FUNCTION_BLOCK FB_CartCtrlStandColuAdjust EXTENDS FB_CartCtrlBase
VAR_INPUT
END_VAR
VAR_OUTPUT
END_VAR
VAR

	m_actJntPos: Vec8d;
	m_tarJntPos : LREAL;
	m_trjJntPos : LREAL;
	m_trjJntInc : LREAL;
	m_lastTrajJntPos : LREAL;
	m_initActJntPos: LREAL;
	m_maxJntPos : vec8d;

	// time threshold to 5-8joint after it's enabled
	m_cartAdjustStartWaitTime :LREAL := 0.3;
	
	//adjust start  time 
	m_adjustStartTime :LREAL;
	m_jntOTG : FB_secOrdTrajFilter;
	
	// filter cut-off frequency for joint 3 velocity
	m_cmdJoystickLpfJnt3Freq : LREAL :=8;
	m_cartCtrlFreq :LREAL:=8000;
END_VAR

// override this function in each exact controller
METHOD PROTECTED calcCmdJntPos : BOOL
VAR_IN_OUT CONSTANT
	// slave cart joint data
	i_slaveCart :FB_SlaveCart;
END_VAR

VAR
	i:INT;
END_VAR
//In this method, 5 represents the pillar postion , 6 represents the beam rotation angle ,7 represents the beam stretch position ,8 represents the overhang angle
m_adjustStartTime :=LIMIT(0, m_adjustStartTime + g_cartCtrlCycleTime, 1);
m_actJntPos := i_slaveCart.curJntPos;
m_jntEnableFlag[5] := BOOL_TO_INT( NOT SafetyCheck.m_safetyCheckData.m_cartStandColumnErr);

IF m_adjustStartTime > m_cartAdjustStartWaitTime THEN
	m_trjJntInc := m_trjJntInc + (i_slaveCart.m_columnJntVel * g_cartCtrlCycleTime);
	m_trjJntPos := m_initActJntPos + m_trjJntInc;
	m_jntPosReachLimit[5] := calcCmdReachLimit();
	m_tarJntPos := LIMIT(GVL_CartMotorParameters.g_minJntPos[5] + GVL_CartControlParameters.g_carJntSoftwareLimit[5], m_trjJntPos, MAX(m_actJntPos[5],i_slaveCart.m_cartDataFromUI.m_standColumnHightLimit));
	m_jntOTG.run(i_targetPos:= m_tarJntPos, i_targetVel:= 0.0, o_cmdAcc=> , o_cmdVel=> , o_cmdPos=>m_cmdJntPos[5] );
END_IF
END_METHOD

METHOD calcCmdReachLimit : BOOL
VAR_INPUT
END_VAR

VAR
	i : INT;
END_VAR

IF (GVL_CartMotorParameters.g_minJntPos[5] + GVL_CartControlParameters.g_carJntSoftwareLimit[5]) >= m_trjJntPos THEN
	IF (m_trjJntInc - m_lastTrajJntPos) <0 THEN
		m_trjJntInc := m_lastTrajJntPos;
	END_IF
	calcCmdReachLimit := TRUE;

ELSIF m_trjJntPos>=(m_maxJntPos[5] - GVL_CartControlParameters.g_carJntSoftwareLimit[5]) THEN
	IF (m_trjJntInc - m_lastTrajJntPos) >0 THEN
		m_trjJntInc := m_lastTrajJntPos;
	END_IF
	calcCmdReachLimit := TRUE;
END_IF
m_lastTrajJntPos := m_trjJntInc;
END_METHOD

// override this function in each exact controller
// NOTICE: set joint control mode here, and do some initialization if needed
METHOD PUBLIC init : BOOL
VAR_IN_OUT CONSTANT
	i_slaveCart	:FB_SlaveCart;
END_VAR
VAR_IN_OUT 
	r_cartCtrlCmd :ST_SlaveArmCtrlCmds;
END_VAR
VAR
	i:INT;
END_VAR
// check if to hold the command joint position unchanged
//m_holdLastCmds := checkToHoldLastCmds(i_slaveCart);
m_holdLastCmds := checkToHoldLastCmds(i_slaveCart);
SUPER^.init(i_slaveCart,r_cartCtrlCmd);
m_cmdJntPos[5]:=i_slaveCart.m_curJntPos[5];

m_jntEnableFlag[5] := BOOL_TO_INT( NOT SafetyCheck.m_safetyCheckData.m_cartStandColumnErr);
m_jntOPMode[5]:= DriverOPMode_cspMZ;
IF GVL_interactUI.g_heightLimitEnbale=FALSE THEN
	m_maxJntPos[5] := i_slaveCart.m_cartDataFromUI.m_standColumnHightLimit;
ELSE
	m_maxJntPos[5] := i_slaveCart.m_cartDataFromUI.m_standColumnHightLimit + GVL_CartControlParameters.g_carJntSoftwareLimit[5];
END_IF
m_initActJntPos:=m_cmdJntPos[5];
m_jntOTG.init(i_curCmdPos:= m_cmdJntPos[5], i_curCmdVel:= 0, i_maxV:=GVL_CartControlParameters.g_maxJntVel[5] , i_maxA:=GVL_CartControlParameters.g_maxJntAcc[5] , i_Ts:=g_cartCtrlCycleTime );

m_trjJntInc := 0;
m_lastTrajJntPos := 0;
m_adjustStartTime := 0;
// update commands to arm
copyCmds(r_cartCtrlCmd);
END_METHOD

END_FUNCTION_BLOCK

(* stored: Version 1.1.0.1, ProductVersion 3.1.4024.11
   POU FB_CartCtrlStandColuAdjust: Id {77449265-3720-4348-92be-3587ec5b4bd0}, SpecialFunc None
   Method calcCmdJntPos: Id {32e8a7e7-7ce7-47cc-b735-666ef264f588}
   Method calcCmdReachLimit: Id {22f72dc3-8b19-4025-9a48-dee178e11d4a}
   Method init: Id {4e005dd2-b8f8-43fd-9139-96a55ce5d52f} *)
